FUNCTION_BLOCK SawmillModule
  (* Standard: 61499-2 *)
  (* Version 0.1, 2017-00-16, hpea485, UOA *)
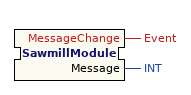
  EVENT_OUTPUT
    MessageChange;
  END_EVENT
  VAR_OUTPUT
    Message : INT;
  END_VAR
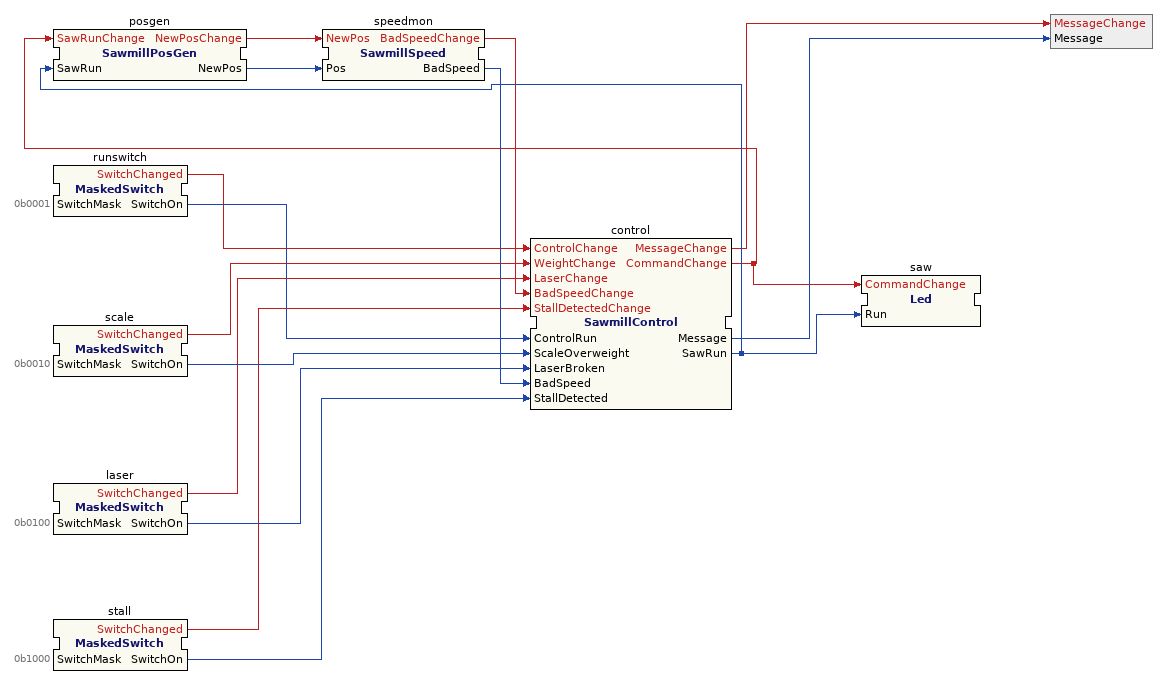
  FBS
    saw : Led;
    control : SawmillControl;
    runswitch : MaskedSwitch(SwitchMask := 0b0001);
    scale : MaskedSwitch(SwitchMask := 0b0010);
    laser : MaskedSwitch(SwitchMask := 0b0100);
    speedmon : SawmillSpeed;
    posgen : SawmillPosGen;
    stall : MaskedSwitch(SwitchMask := 0b1000);
  END_FBS
  EVENT_CONNECTIONS
    control.MessageChange TO MessageChange;
    control.CommandChange TO saw.CommandChange;
    control.CommandChange TO posgen.SawRunChange;
    runswitch.SwitchChanged TO control.ControlChange;
    scale.SwitchChanged TO control.WeightChange;
    laser.SwitchChanged TO control.LaserChange;
    speedmon.BadSpeedChange TO control.BadSpeedChange;
    posgen.NewPosChange TO speedmon.NewPos;
    stall.SwitchChanged TO control.StallDetectedChange;
  END_CONNECTIONS
  DATA_CONNECTIONS
    control.Message TO Message;
    control.SawRun TO saw.Run;
    control.SawRun TO posgen.SawRun;
    runswitch.SwitchOn TO control.ControlRun;
    scale.SwitchOn TO control.ScaleOverweight;
    laser.SwitchOn TO control.LaserBroken;
    speedmon.BadSpeed TO control.BadSpeed;
    posgen.NewPos TO speedmon.Pos;
    stall.SwitchOn TO control.StallDetected;
  END_CONNECTIONS
END_FUNCTION_BLOCK
